{attribute 'qualified_only'}
{attribute 'strict'}
TYPE SortOrder :
(
	ASCENDING,
	DESCENDING
);
END_TYPE

(* stored: Version 1.1.0.1, ProductVersion 3.1.4024.12
   EnumerationTextList SortOrder: Id {00d7a571-b6f2-0d82-23f6-8206b5c22cc7} *)
